// TIA Portal V17 export
// export: Created 2021-12-03T08:08:02.120089Z, ExportSetting WithDefaults, DisplayName Totally Integrated Automation Portal, DisplayVersion V17, DisplayName TIA Portal Openness, DisplayVersion V17, DisplayName TIA Portal Version Control Interface, DisplayVersion V17, DisplayName STEP 7 Professional, DisplayVersion V17, DisplayName STEP 7 Safety, DisplayVersion V17, DisplayName WinCC Advanced, DisplayVersion V17
VAR_GLOBAL   // PLC tag table "DetLine"
   DetLineSts_Sts AT %MW15 : Word;
   DetLineSts_ConOk AT %M15.0 : Bool;
   DetLineSts_SyncStrt AT %M15.1 : Bool;
   DetLineSts_ScanAct AT %M15.2 : Bool;
   DetLineSts_RdyForScan AT %M15.3 : Bool;
   DetLineSnd_ScanData AT %MW17 : Word;
   DetLineSnd_HighDose AT %M17.0 : Bool;
   DetLineSnd_Direct AT %M17.1 : Bool;
END_VAR
